# EPICS substitutions: viocs/ts_bpms/ts_bpmsApp/Db/bpm.substitutions
file "db/bpm.db" {
    pattern { sector, pos }

        { "01", "" }
        { "02", "" }
        { "03", "" }
        { "04", "-A" }
        { "04", "-B" }
}
